(* PLC project 117_1_V0.5.project, CODESYS CODESYS V3.5 SP17 Patch 3 *)
(* stored: creationDateTime 1970-01-01T00:00:00, modificationDateTime 2026-03-26T18:14:32.4070562 *)

FUNCTION_BLOCK OutputManager
  VAR
    OutputBytes : ARRAY[0..1] OF BYTE;
    bitsOutput : ARRAY[0..15] OF BOOL;
    iByte : INT;
    iBit : INT;
    tempByte : BYTE;
  END_VAR

            FOR iByte := 0 TO 1 DO
    tempByte := 0;
    FOR iBit := 0 TO 7 DO
        tempByte := tempByte OR (SEL(bitsOutput[iByte*8 + iBit], 0,SHL(BYTE#16#01,iBit)));
    END_FOR
    OutputBytes[iByte] := tempByte;
END_FOR
          

METHOD set_data : BOOL
  VAR_INPUT
    varName : DQ_VARS;
    enable : BOOL := FALSE;
  END_VAR
                  bitsOutput[varName]:= enable;
set_data := bitsOutput[varName];
                
END_METHOD
END_FUNCTION_BLOCK
